// TIA Portal V18 export
// export: Created 2025-12-01T17:51:25.1965133Z, ExportSetting None, DisplayName Totally Integrated Automation Portal, DisplayVersion V18 Update 5, DisplayName TIA Portal Openness, DisplayVersion V18 Update 5, DisplayName TIA Portal Teamcenter Gateway, DisplayVersion V18, DisplayName TIA Portal Version Control Interface, DisplayVersion V18, DisplayName STEP 7 Professional, DisplayVersion V18 Update 5, DisplayName STEP 7 Safety, DisplayVersion V18, DisplayName WinCC Professional, DisplayVersion V18 Update 5
DATA_BLOCK "NG_DB"   // DB2901
// stored: AutoNumber false, InstanceOfName NG, InstanceOfType FB
"NG"
   // VAR
   //    NG_L_1 : "NGStatus";
   //    NG_L_2 { S7_SetPoint := 'True'} : "NGStatus";
   //    NG_L_3 { S7_SetPoint := 'True'} : "NGStatus";
   //    NG_UL_1 { S7_SetPoint := 'True'} : "NGStatus";
   //    NG_UL_2 { S7_SetPoint := 'True'} : "NGStatus";
   //    NG_UL_3 { S7_SetPoint := 'True'} : "NGStatus";
   // END_VAR
BEGIN
END_DATA_BLOCK
